FUNCTION_BLOCK HydraulicMotor
VAR_INPUT
	par : ST_pValveControlledCylinder;
	PressureIn : LREAL;
	PressureOut : LREAL;
END_VAR
VAR_OUTPUT
	Torque : LREAL;
END_VAR
VAR
	dpsum : LREAL;					//[pa]
	Dm : LREAL := 189;				//[cm^3/Rev]
	nhm : LREAL := 0.9;			//[-]
END_VAR

//For controlling the king joint, aka rotation of the whole crane horisontally
//dpsum = (PressureIn - PressureOut);

dpsum := (PressureIn - PressureOut);

Torque := ( dpsum * Dm * nhm * EXPT(10,(-6))) / (2 * par.pi);

END_FUNCTION_BLOCK

(* stored: Version 1.1.0.1, ProductVersion 3.1.4024.9
   POU HydraulicMotor: Id {90f53dd3-8e70-4d35-83cf-1af75a7a3a25}, SpecialFunc None *)
